// TIA Portal project "Practica_Motor_Trifasica" (V16)

(* hardware
DEVICE "S7-1200 station_1"  S7-1200 Station
   slot 0: "Rack_0"  S7-1200 Rack  Rack  V1.0
   slot 1: "PLC_1"  CPU 1214C AC/DC/Rly  6ES7 214-1BE30-0XB0  V2.2
*)

// ===== PLC "PLC_1"  CPU 1214C AC/DC/Rly =====

VAR_GLOBAL   // PLC tag table "Tabla de variables estándar"
   "Encendido" AT %I0.0 : Bool;
   "Stop" AT %I0.1 : Bool;
   "Cambio" AT %I0.2 : Bool;
   "KM1" AT %Q0.0 : Bool;
   "KM2" AT %Q0.1 : Bool;
   "KM3" AT %Q0.2 : Bool;
   "M0" AT %M0.0 : Bool;
END_VAR

// folder: System blocks/Program resources

DATA_BLOCK "IEC_Timer_0_DB_2"   // DB3
{ S7_Optimized_Access := 'TRUE' }
AUTHOR : Simatic
FAMILY : IEC
NAME : IEC_TMR
VERSION : 1.0
// stored: InstanceOfName IEC_TIMER
"IEC_TIMER"
BEGIN
END_DATA_BLOCK

DATA_BLOCK "IEC_Timer_0_DB_3"   // DB4
{ S7_Optimized_Access := 'TRUE' }
AUTHOR : Simatic
FAMILY : IEC
NAME : IEC_TMR
VERSION : 1.0
// stored: InstanceOfName IEC_TIMER
"IEC_TIMER"
BEGIN
END_DATA_BLOCK

// folder: (top level)

ORGANIZATION_BLOCK "Main"   // OB1, LAD, ProgramCycle
TITLE = "Main Program Sweep (Cycle)"
{ S7_Optimized_Access := 'TRUE' }
VERSION : 0.1
BEGIN

REGION Network 1
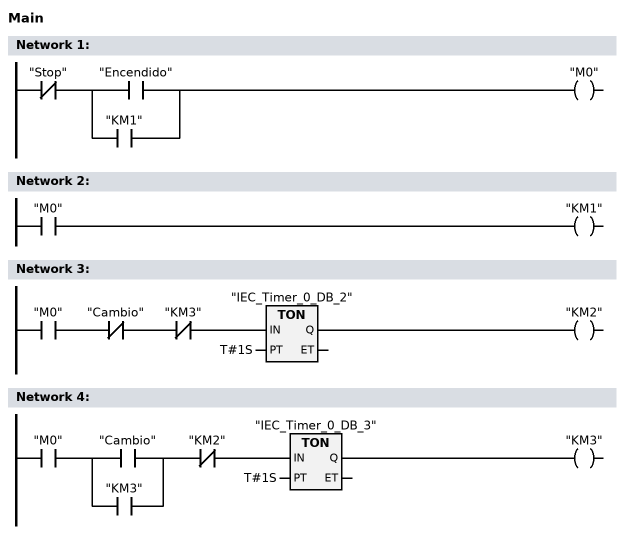
   RUNG wire#powerrail
      I_Contact( "Stop" )
      wire#w1
      Contact( "Encendido" )
      wire#w2
      Coil( "M0" )
   END_RUNG
   RUNG wire#w1
      Contact( "KM1" )
   END_RUNG wire#w2
   // the same network as SCL:
   "M0" := NOT "Stop" AND ("Encendido" OR "KM1");
END_REGION

REGION Network 2
   RUNG wire#powerrail
      Contact( "M0" )
      Coil( "KM1" )
   END_RUNG
   // the same network as SCL:
   "KM1" := "M0";
END_REGION

REGION Network 3
   "IEC_Timer_0_DB_2".TON(IN := "M0" AND NOT "Cambio" AND NOT "KM3", PT := T#1S);
   "KM2" := "IEC_Timer_0_DB_2".Q;
END_REGION

REGION Network 4
   "IEC_Timer_0_DB_3".TON(IN := "M0" AND ("Cambio" OR "KM3") AND NOT "KM2", PT := T#1S);
   "KM3" := "IEC_Timer_0_DB_3".Q;
END_REGION
END_ORGANIZATION_BLOCK